RoboDK station: rdk_prog.rdk

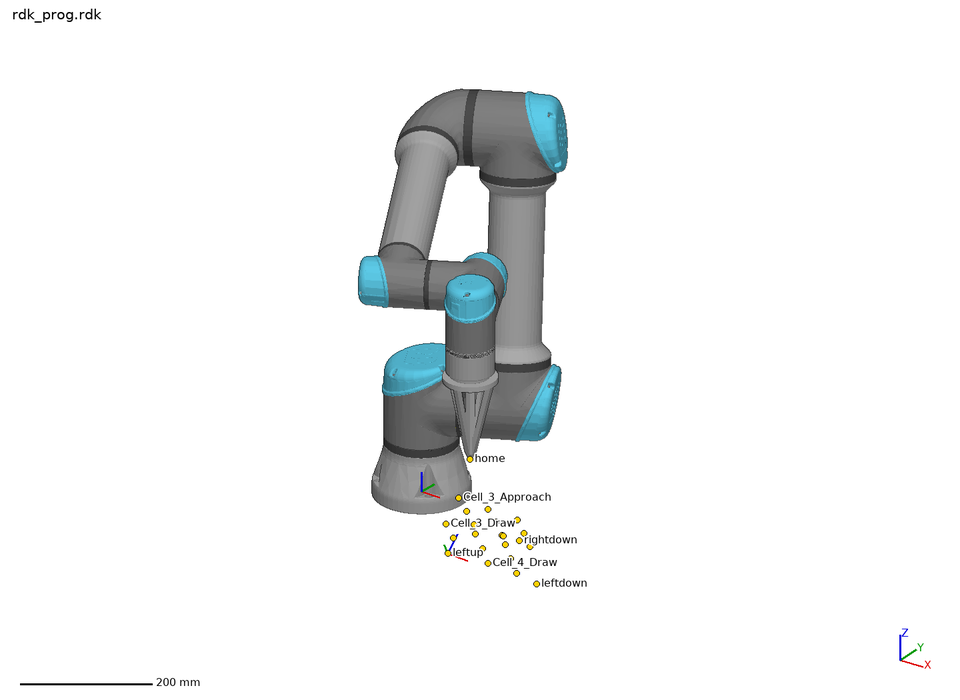
[picture v0: the station drawn from its stored meshes, robots at their saved joint values, targets as dots, program paths as lines]
Station tic-tac-toe (saved by RoboDK 6.0.3). Poses are relative to the parent item; angles as X-Y-Z fixed-axis rotations.
  - frame UR5e Base at (0, 0, 0) mm
    - robot UR5e: 6 axes, payload 5 kg, reach 850 mm, repeatability 0.03 mm, weight 18.4 kg
        modified DH rows (alpha deg, a mm, theta deg, d mm): 0, 0, 0, 162.5; 90, 0, 180, 0; 0, 425, 0, 0; 0, 392.25, 0, 133.3; -90, 0, 0, 99.7; 90, 0, 180, 99.6
        joint limits [-360, -360, -360, -360, -360, -360] to [360, 360, 360, 360, 360, 360]; home [0, -90, -90, 0, 90, 0]; saved at [116.688, -100.979, 112.736, -101.756, -90, -153.312]
      - tool Marker, TCP at (0, 0, 100) mm
      - tool tool, TCP at (0, 0, 141.6) mm, size 85 x 141.5 x 85 mm, geometry from tool.stl
    - target leftup (Cartesian target) at (373.48, -463.52, 186.32) mm, rotated rx -171.62 ry -25.21 rz -149.02 deg; joints [-27.537, -105.174, -98.877, -72.059, 64.183, 31.009] of UR5e
    - target leftdown (Cartesian target) at (470.21, -366.55, 123.15) mm, rotated rx -171.68 ry -25.27 rz -149.04 deg; joints [-15.151, -111.906, -98.288, -71.707, 66.128, 44.544] of UR5e
    - target rightdown (Cartesian target) at (364.78, -262.27, 125.11) mm, rotated rx -171.69 ry -25.32 rz -149.03 deg; joints [-6.02, -93.945, -119.941, -71.797, 68.279, 54.166] of UR5e
  - frame board at (373.48, -463.52, 186.32) mm, rotated rx -3.57 ry 26.26 rz 42.02 deg
    - target home (Cartesian target) at (17.24, 164.78, 99.56) mm, rotated rx -159.1 ry -16.64 rz -45.95 deg; joints [116.688, -100.979, 112.736, -101.756, -90, -153.312] of UR5e
    - target Cell_1_Draw (Cartesian target) at (25, 25, 0) mm, rotated rx -180 ry 0 rz 0 deg; joints [128.078, -75.468, 105.177, -125.612, -115.862, -186.134] of UR5e
    - target Cell_2_Draw (Cartesian target) at (20, 72.5, 2.5) mm, rotated rx -180 ry 0 rz 0 deg; joints [127.164, -81.582, 112.644, -127.404, -115.765, 172.856] of UR5e
    - target Cell_3_Draw (Cartesian target) at (15, 120, 4) mm, rotated rx -180 ry 0 rz 0 deg; joints [125.999, -87.913, 119.721, -128.707, -115.63, 171.571] of UR5e
    - target Cell_4_Draw (Cartesian target) at (72, 25, 1) mm, rotated rx -180 ry 0 rz 0 deg; joints [132.506, -73.278, 104.99, -125.456, -116.235, -181.223] of UR5e
    - target Cell_5_Draw (Cartesian target) at (70, 75, 3.5) mm, rotated rx 180 ry 0 rz 0 deg; joints [132.319, -79.356, 112.887, -127.367, -116.222, 178.57] of UR5e
    - target Cell_6_Draw (Cartesian target) at (65, 122.5, 6) mm, rotated rx -180 ry 0 rz 0 deg; joints [131.762, -85.567, 119.929, -128.472, -116.184, 177.95] of UR5e
    - target Cell_7_Draw (Cartesian target) at (120, 25, 2.5) mm, rotated rx -180 ry 0 rz 0 deg; joints [136.962, -70.645, 104.093, -124.987, -116.44, 183.744] of UR5e
    - target Cell_8_Draw (Cartesian target) at (117.5, 75, 5) mm, rotated rx -180 ry 0 rz 0 deg; joints [137.161, -76.507, 112.003, -126.937, -116.445, -176.033] of UR5e
    - target Cell_9_Draw (Cartesian target) at (115, 125, 7) mm, rotated rx 180 ry 0 rz 0 deg; joints [137.376, -82.52, 119.434, -128.248, -116.451, -175.794] of UR5e
    - target Cell_1_Approach (Cartesian target) at (25, 25, 50) mm, rotated rx 180 ry 0 rz 0 deg; joints [130.372, -78.209, 101.064, -117.645, -116.076, 176.406] of UR5e
    - target Cell_2_Approach (Cartesian target) at (20, 72.5, 50) mm, rotated rx -180 ry 0 rz 0 deg; joints [129.551, -84.418, 108.561, -119.333, -116.005, 175.496] of UR5e
    - target Cell_3_Approach (Cartesian target) at (15, 120, 50) mm, rotated rx -180 ry 0 rz 0 deg; joints [128.554, -90.873, 115.536, -120.336, -115.91, 174.392] of UR5e
    - target Cell_4_Approach (Cartesian target) at (72, 25, 50) mm, rotated rx -180 ry 0 rz 0 deg; joints [134.74, -75.963, 100.95, -117.629, -116.359, 181.265] of UR5e
    - target Cell_5_Approach (Cartesian target) at (70, 75, 50) mm, rotated rx -180 ry 0 rz 0 deg; joints [134.65, -82.148, 108.871, -119.409, -116.355, 181.165] of UR5e
    - target Cell_6_Approach (Cartesian target) at (65, 122.5, 50) mm, rotated rx -180 ry 0 rz 0 deg; joints [134.2, -88.409, 115.895, -120.395, -116.333, 180.663] of UR5e
    - target Cell_7_Approach (Cartesian target) at (120, 25, 50) mm, rotated rx -180 ry 0 rz 0 deg; joints [139.09, -73.225, 100.175, -117.43, -116.478, 186.121] of UR5e
    - target Cell_8_Approach (Cartesian target) at (117.5, 75, 50) mm, rotated rx -180 ry 0 rz 0 deg; joints [139.369, -79.191, 108.123, -119.274, -116.48, 186.433] of UR5e
    - target Cell_9_Approach (Cartesian target) at (115, 125, 50) mm, rotated rx -180 ry 0 rz 0 deg; joints [139.707, -85.303, 115.497, -120.367, -116.481, 186.81] of UR5e
    - target Target 20 (Cartesian target) at (75, 25, 50) mm, rotated rx 180 ry 0 rz 0 deg; joints [135.27, 19.295, 261.337, -13.012, -116.382, 191.856] of UR5e
    - target Target 21 (Cartesian target) at (25, 25, 50) mm, rotated rx 180 ry 0 rz 0 deg; joints [130.372, -78.209, 101.064, -117.645, -116.076, 176.406] of UR5e
  - program Prog1 (3 instructions, listed below)

--- program Prog1 (robot UR5e) ---
  Set Ref.: board
  Set Tool: tool
  MoveL (home)
